// Mitsubishi GX Works2 project: EexcB-group13-1 (1) (1)   PLC: FX3G

// global labels: Global1
VAR_GLOBAL
  Switch7 AT X007 : BOOL;
  WorkLight AT Y007 : BOOL;
  Emergency_button AT X005 : BOOL;
  RaspberryStock AT D1100 : REAL;
  RaspberryInput AT D1110 : REAL;
  LemonStock AT D1102 : REAL;
  LemonInput AT D1112 : REAL;
  GummyBearStock AT D1104 : REAL;
  GummyBearInput AT D1114 : REAL;
  StablilizingMaterialStock AT D1106 : REAL;
  StablilizingMaterialInput AT D1116 : REAL;
  ANALOG_INPUT AT D8280 : INT;
  Intialize_produce AT X001 : BOOL;
  REGULAR_ICECREAM AT M0 : BOOL;
  ICE_CREAM_TYPE AT D1108 : REAL;
  UNDER_5 AT M2 : BOOL;
  UPPER_0 AT M3 : BOOL;
  UNDER_10 AT M4 : BOOL;
  UPPER_6 AT M6 : BOOL;
  PINUK_ICECREAM AT M1 : BOOL;
  LEMON_PINUK AT M11 : BOOL;
  RASPBERRY_PINUK AT M12 : BOOL;
  StABILIZE_PINUK AT M13 : BOOL;
  GUMMYBEAR_PINUK AT M14 : BOOL;
  RASPBERRY_REGUKAR AT M15 : BOOL;
  LEMON_REGULAR AT M16 : BOOL;
  StABILIZE_REGULAR AT M17 : BOOL;
  GUMMYBEAR_REGULAR AT M18 : BOOL;
  ICECREAM_APPROVE AT M19 : BOOL;
  TIMER_LIGHT_MIX AT TC0 : BOOL;
  LIGHT_TIMER_SWITCH AT TS0 : BOOL;
  LIGHT_TIMER_SWITCH_Y0 AT TS0 : BOOL;
  MAKING_LIGHT AT Y000 : BOOL;
  MAKING_TIMER_SWITCH_Y0 AT TS0 : BOOL;
  MAKING_TIMER AT TC0 : BOOL;
  MAKING_PROCESS AT M30 : BOOL;
  MOVE_TO_FREEZE_SWITCH AT X002 : BOOL;
  LEMON_MAKE_CONTAINER AT M21 : BOOL;
  RASPBERRY_MAKE_CONTAINER AT M22 : BOOL;
  FREEZE_LIGHT AT Y002 : BOOL;
  FREEZE_process AT M25 : BOOL;
  FREEZING_TIMER AT TC1 : BOOL;
  SENSOR_10 AT X003 : BOOL;
  FREEZING_TIMER_SWITCH AT TS1 : BOOL;
  FREEZE_DONE AT M26 : BOOL;
  MIX_PROCESS AT M26 : BOOL;
  MIX_CONTAINER AT M27 : BOOL;
  PINUK_MIX_TIMER AT TC2 : BOOL;
  REGULAR_MIX_TIMER AT TC3 : BOOL;
  PINUK_MIX_SWITCH AT TS2 : BOOL;
  REGULAR_MIX_SWITCH AT TS3 : BOOL;
  START_MIX AT M28 : BOOL;
  MIX_LIGHT_TIMER_1 AT TC4 : BOOL;
  MIX_LIGHT_SWITCH_1 AT TS4 : BOOL;
  BLINK_ENABLE AT M29 : BOOL;
  MIX_LIGHT_TIMER_2 AT TC5 : BOOL;
  MIX_LIGHT_SWITCH_2 AT TS5 : BOOL;
  TYPE_CHOSEN AT M10 : BOOL;
  ICECREAM_counter AT CC0 : BOOL;
  ICECREAM_READY AT M31 : BOOL;
  PROCESS_DONE AT M32 : BOOL;
  ANALOG_OUTPUT AT D8282 : INT;
  Sop AT M33 : BOOL;
  OUT_OF_STOCK AT M5 : BOOL;
  UNDER_6 AT M34 : BOOL;
  UPPER_5 AT M35 : BOOL;
  BLINK_LIGHT_1 AT Y005 : BOOL;
  BLINK_LIGHT_2 AT Y006 : BOOL;
  DELETE AT X030 : BOOL;
  InVENTORY_CHECK AT M36 : BOOL;
  OUT_OF_RAS AT M37 : BOOL;
  OUT_OF_LEMON AT M38 : BOOL;
  OUT_OF_STABILIZE AT M39 : BOOL;
  OUT_OF_GUMMY AT M40 : BOOL;
  InVENTORY_CHECK_DONE AT M41 : BOOL;
  ICE_CREAM_packs AT D1118 : REAL;
  RASPBERRY_ICECREAM_MAK_CONTAINER AT D1122 : REAL;
  LEMON_ICECREAM_MAK_CONTAINER AT D1120 : REAL;
  LEMON_FREEZE_CONTAINERR AT D1124 : REAL;
  RASPBERRY_FREEZE_CONTAINERR AT D1126 : REAL;
  MIXING_CONTAINER AT D1128 : REAL;
  MOVED_CONTAINER_2 AT M42 : BOOL;
  FINISHED_MOVE_2 AT M43 : BOOL;
  MOVE_CONTAINAER_2 AT TC6 : BOOL;
  FINISH_MOVING_2 AT TS6 : BOOL;
END_VAR

// task Task_01 (event TRUE, interval 0, priority 31): POU_01

PROGRAM POU_01
(* structured ladder/FBD written out as ST: instructions are called as NAME(EN, inputs, outputs); _pN, _eN, _tN stand for wires *)
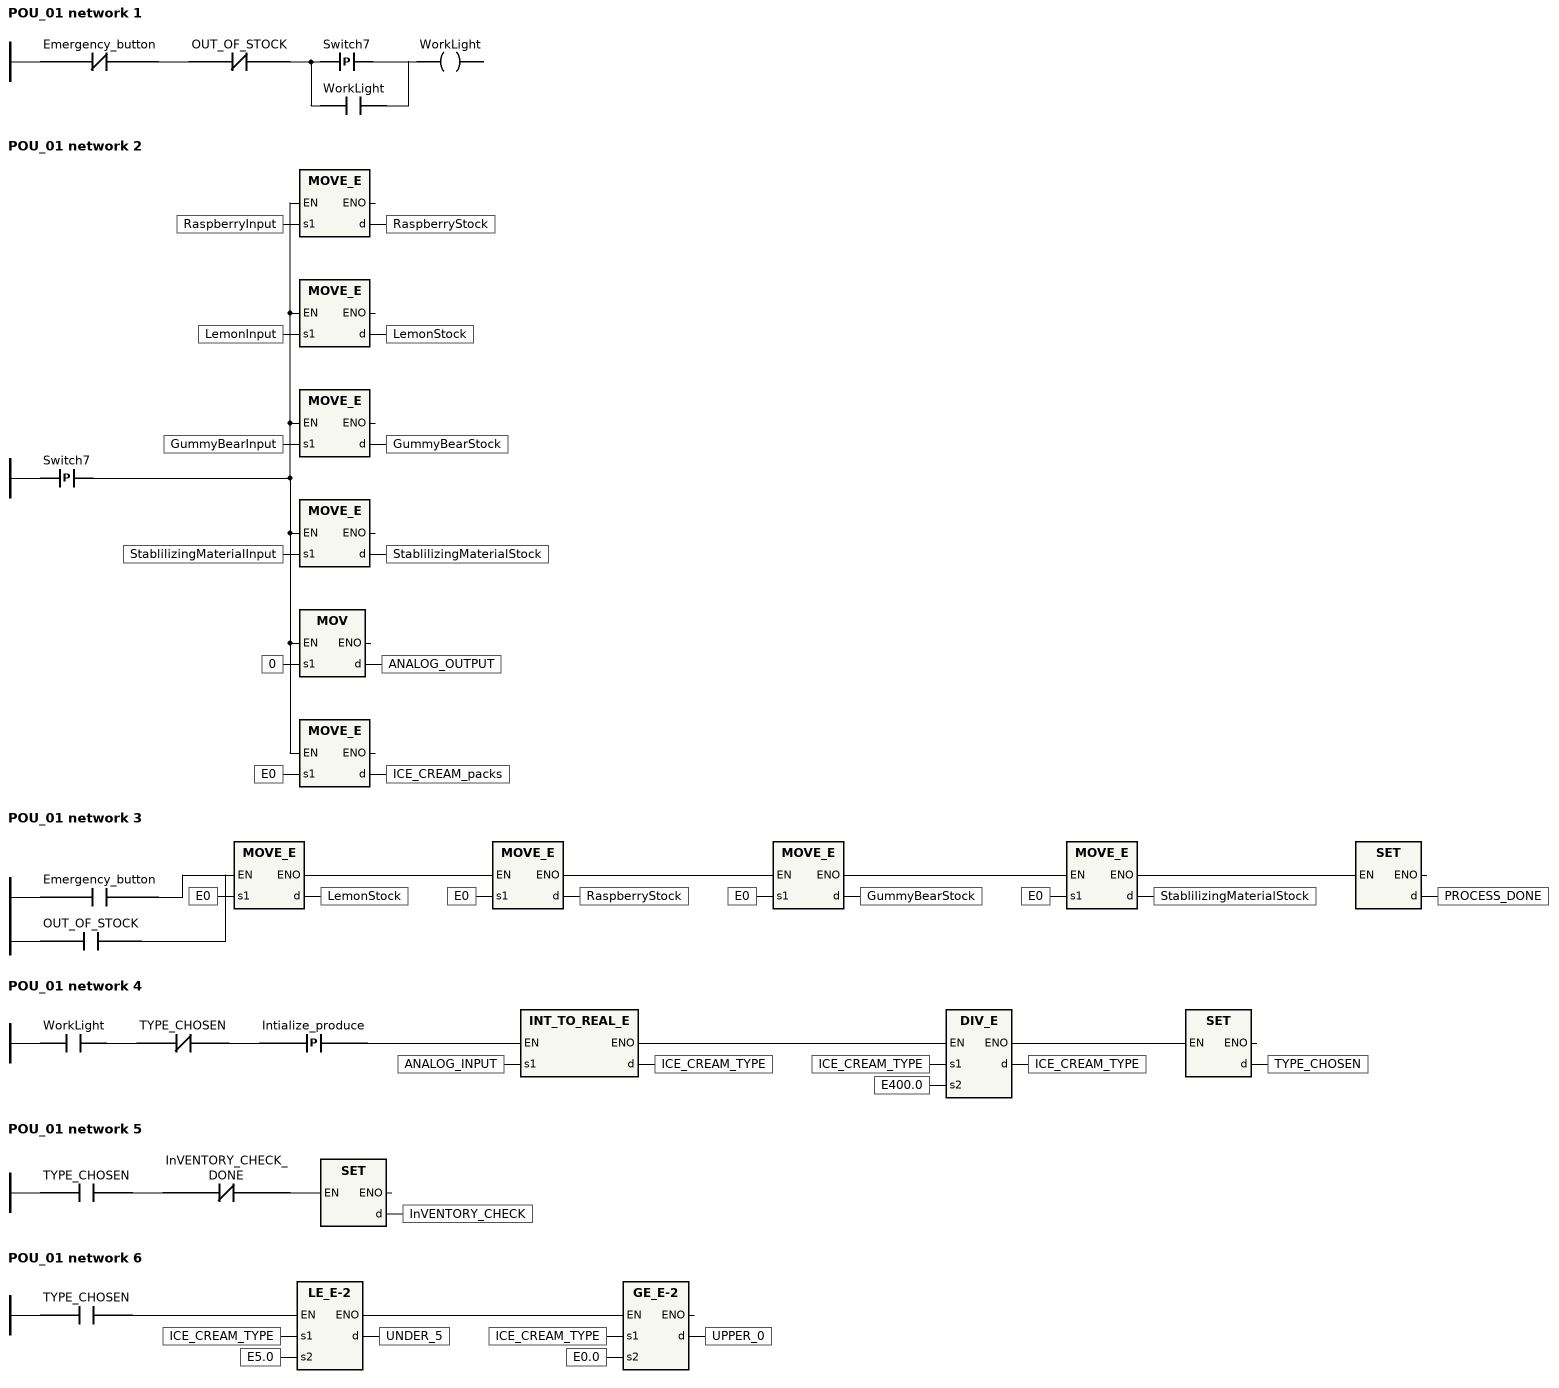
(* network 1 *)
_p1 := NOT Emergency_button AND NOT OUT_OF_STOCK;
WorkLight := (_p1 AND LDP(TRUE, Switch7)) OR (_p1 AND WorkLight);
(* network 2 *)
_p1 := LDP(TRUE, Switch7);
MOVE_E(_p1, RaspberryInput, RaspberryStock);
MOVE_E(_p1, LemonInput, LemonStock);
MOVE_E(_p1, GummyBearInput, GummyBearStock);
MOVE_E(_p1, StablilizingMaterialInput, StablilizingMaterialStock);
MOV(_p1, 0, ANALOG_OUTPUT);
MOVE_E(_p1, E0, ICE_CREAM_packs);
(* network 3 *)
_e1 := MOVE_E(Emergency_button OR OUT_OF_STOCK, E0, LemonStock);
_e2 := MOVE_E(_e1, E0, RaspberryStock);
_e3 := MOVE_E(_e2, E0, GummyBearStock);
_e4 := MOVE_E(_e3, E0, StablilizingMaterialStock);
SET(_e4, PROCESS_DONE);
(* network 4 *)
_e1 := INT_TO_REAL_E(WorkLight AND NOT TYPE_CHOSEN AND LDP(TRUE, Intialize_produce), ANALOG_INPUT, ICE_CREAM_TYPE);
_e2 := DIV_E(_e1, ICE_CREAM_TYPE, E400.0, ICE_CREAM_TYPE);
SET(_e2, TYPE_CHOSEN);
(* network 5 *)
SET(TYPE_CHOSEN AND NOT InVENTORY_CHECK_DONE, InVENTORY_CHECK);
(* network 6 *)
_e1 := LE_E(TYPE_CHOSEN, ICE_CREAM_TYPE, E5.0, UNDER_5);
GE_E(_e1, ICE_CREAM_TYPE, E0.0, UPPER_0);
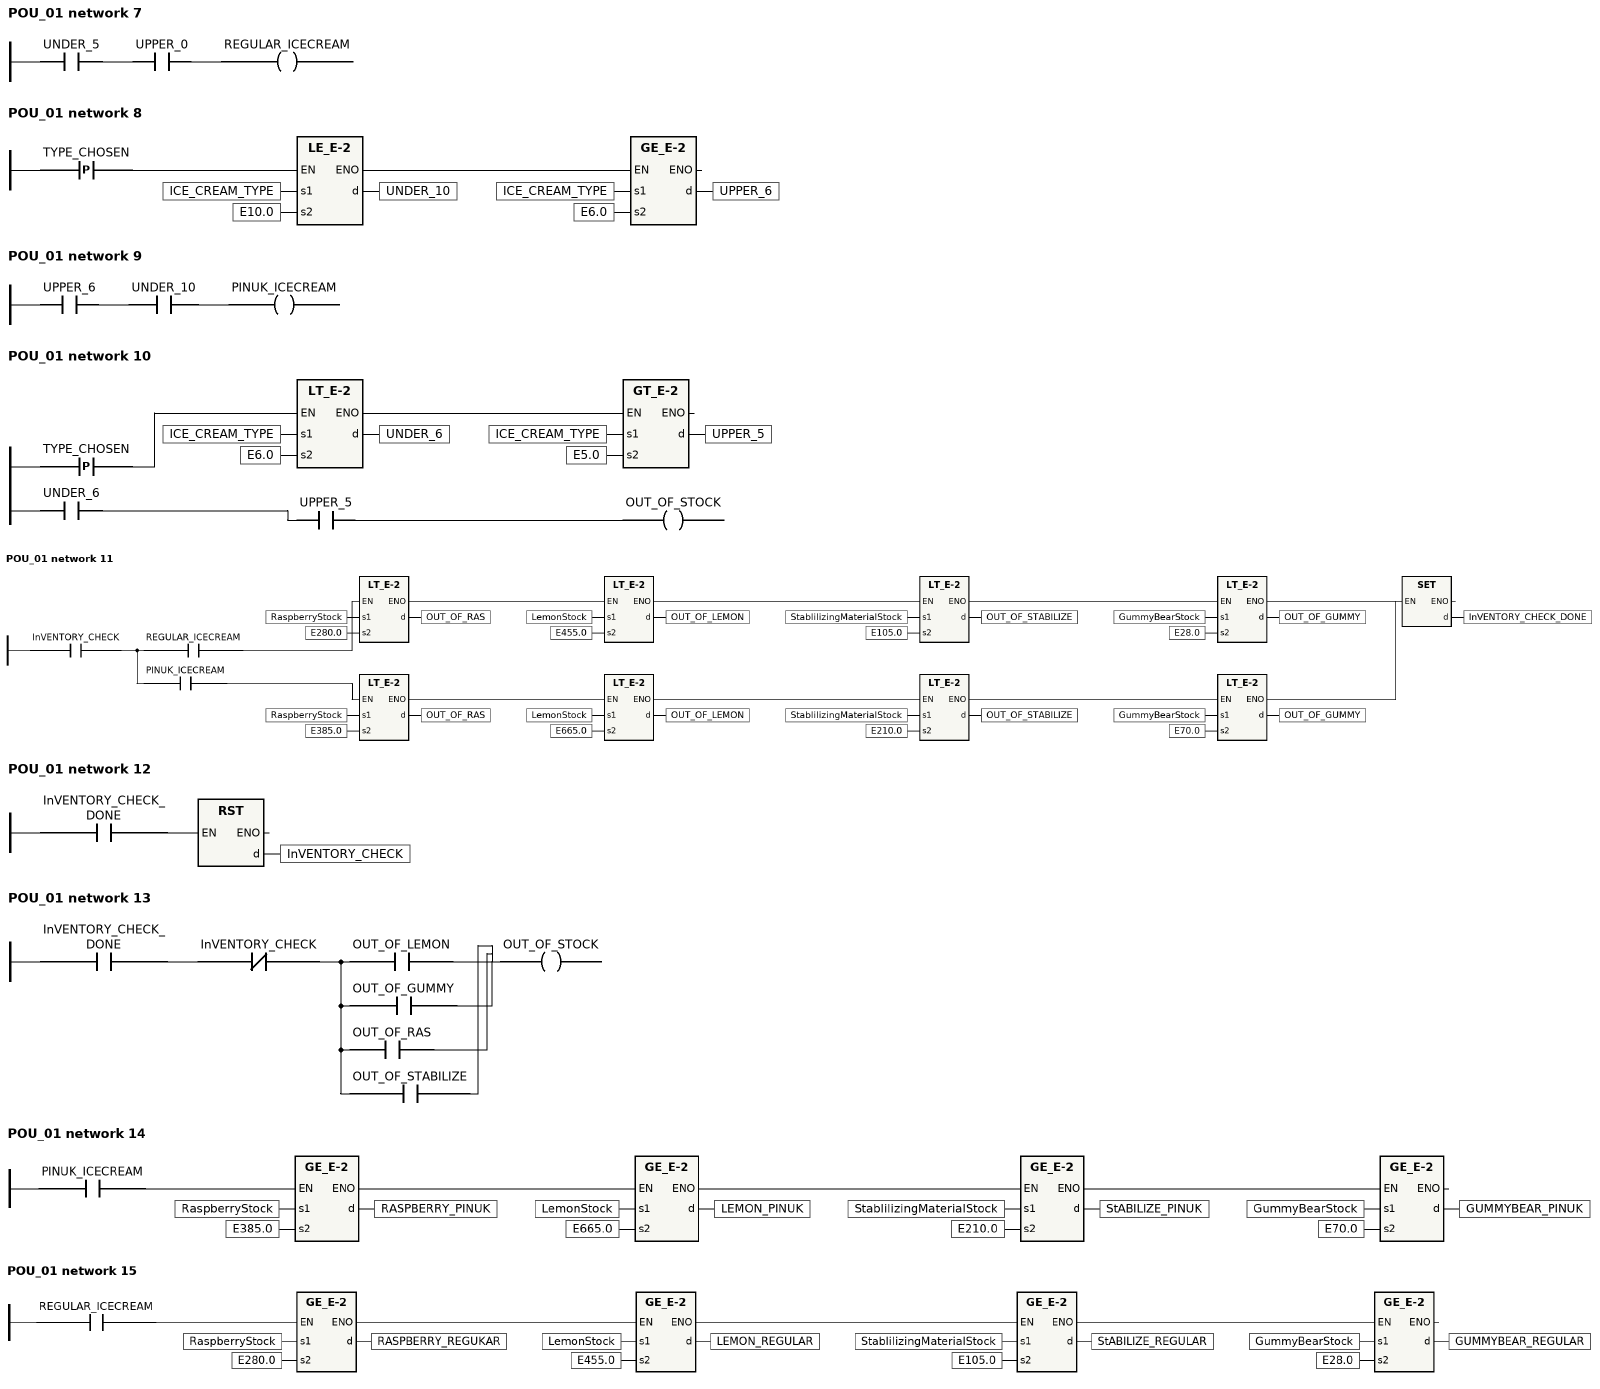
(* network 7 *)
REGULAR_ICECREAM := UNDER_5 AND UPPER_0;
(* network 8 *)
_e1 := LE_E(LDP(TRUE, TYPE_CHOSEN), ICE_CREAM_TYPE, E10.0, UNDER_10);
GE_E(_e1, ICE_CREAM_TYPE, E6.0, UPPER_6);
(* network 9 *)
PINUK_ICECREAM := UPPER_6 AND UNDER_10;
(* network 10 *)
_e1 := LT_E(LDP(TRUE, TYPE_CHOSEN), ICE_CREAM_TYPE, E6.0, UNDER_6);
GT_E(_e1, ICE_CREAM_TYPE, E5.0, UPPER_5);
OUT_OF_STOCK := UNDER_6 AND UPPER_5;
(* network 11 *)
_e1 := LT_E(InVENTORY_CHECK AND REGULAR_ICECREAM, RaspberryStock, E280.0, OUT_OF_RAS);
_e2 := LT_E(_e1, LemonStock, E455.0, OUT_OF_LEMON);
_e3 := LT_E(_e2, StablilizingMaterialStock, E105.0, OUT_OF_STABILIZE);
_e4 := LT_E(_e3, GummyBearStock, E28.0, OUT_OF_GUMMY);
_e5 := LT_E(InVENTORY_CHECK AND PINUK_ICECREAM, RaspberryStock, E385.0, OUT_OF_RAS);
_e6 := LT_E(_e5, LemonStock, E665.0, OUT_OF_LEMON);
_e7 := LT_E(_e6, StablilizingMaterialStock, E210.0, OUT_OF_STABILIZE);
_e8 := LT_E(_e7, GummyBearStock, E70.0, OUT_OF_GUMMY);
SET(_e4 OR _e8, InVENTORY_CHECK_DONE);
(* network 12 *)
RST(InVENTORY_CHECK_DONE, InVENTORY_CHECK);
(* network 13 *)
_p1 := InVENTORY_CHECK_DONE AND NOT InVENTORY_CHECK;
OUT_OF_STOCK := (_p1 AND OUT_OF_LEMON) OR (_p1 AND OUT_OF_GUMMY) OR (_p1 AND OUT_OF_RAS) OR (_p1 AND OUT_OF_STABILIZE);
(* network 14 *)
_e1 := GE_E(PINUK_ICECREAM, RaspberryStock, E385.0, RASPBERRY_PINUK);
_e2 := GE_E(_e1, LemonStock, E665.0, LEMON_PINUK);
_e3 := GE_E(_e2, StablilizingMaterialStock, E210.0, StABILIZE_PINUK);
GE_E(_e3, GummyBearStock, E70.0, GUMMYBEAR_PINUK);
(* network 15 *)
_e1 := GE_E(REGULAR_ICECREAM, RaspberryStock, E280.0, RASPBERRY_REGUKAR);
_e2 := GE_E(_e1, LemonStock, E455.0, LEMON_REGULAR);
_e3 := GE_E(_e2, StablilizingMaterialStock, E105.0, StABILIZE_REGULAR);
GE_E(_e3, GummyBearStock, E28.0, GUMMYBEAR_REGULAR);
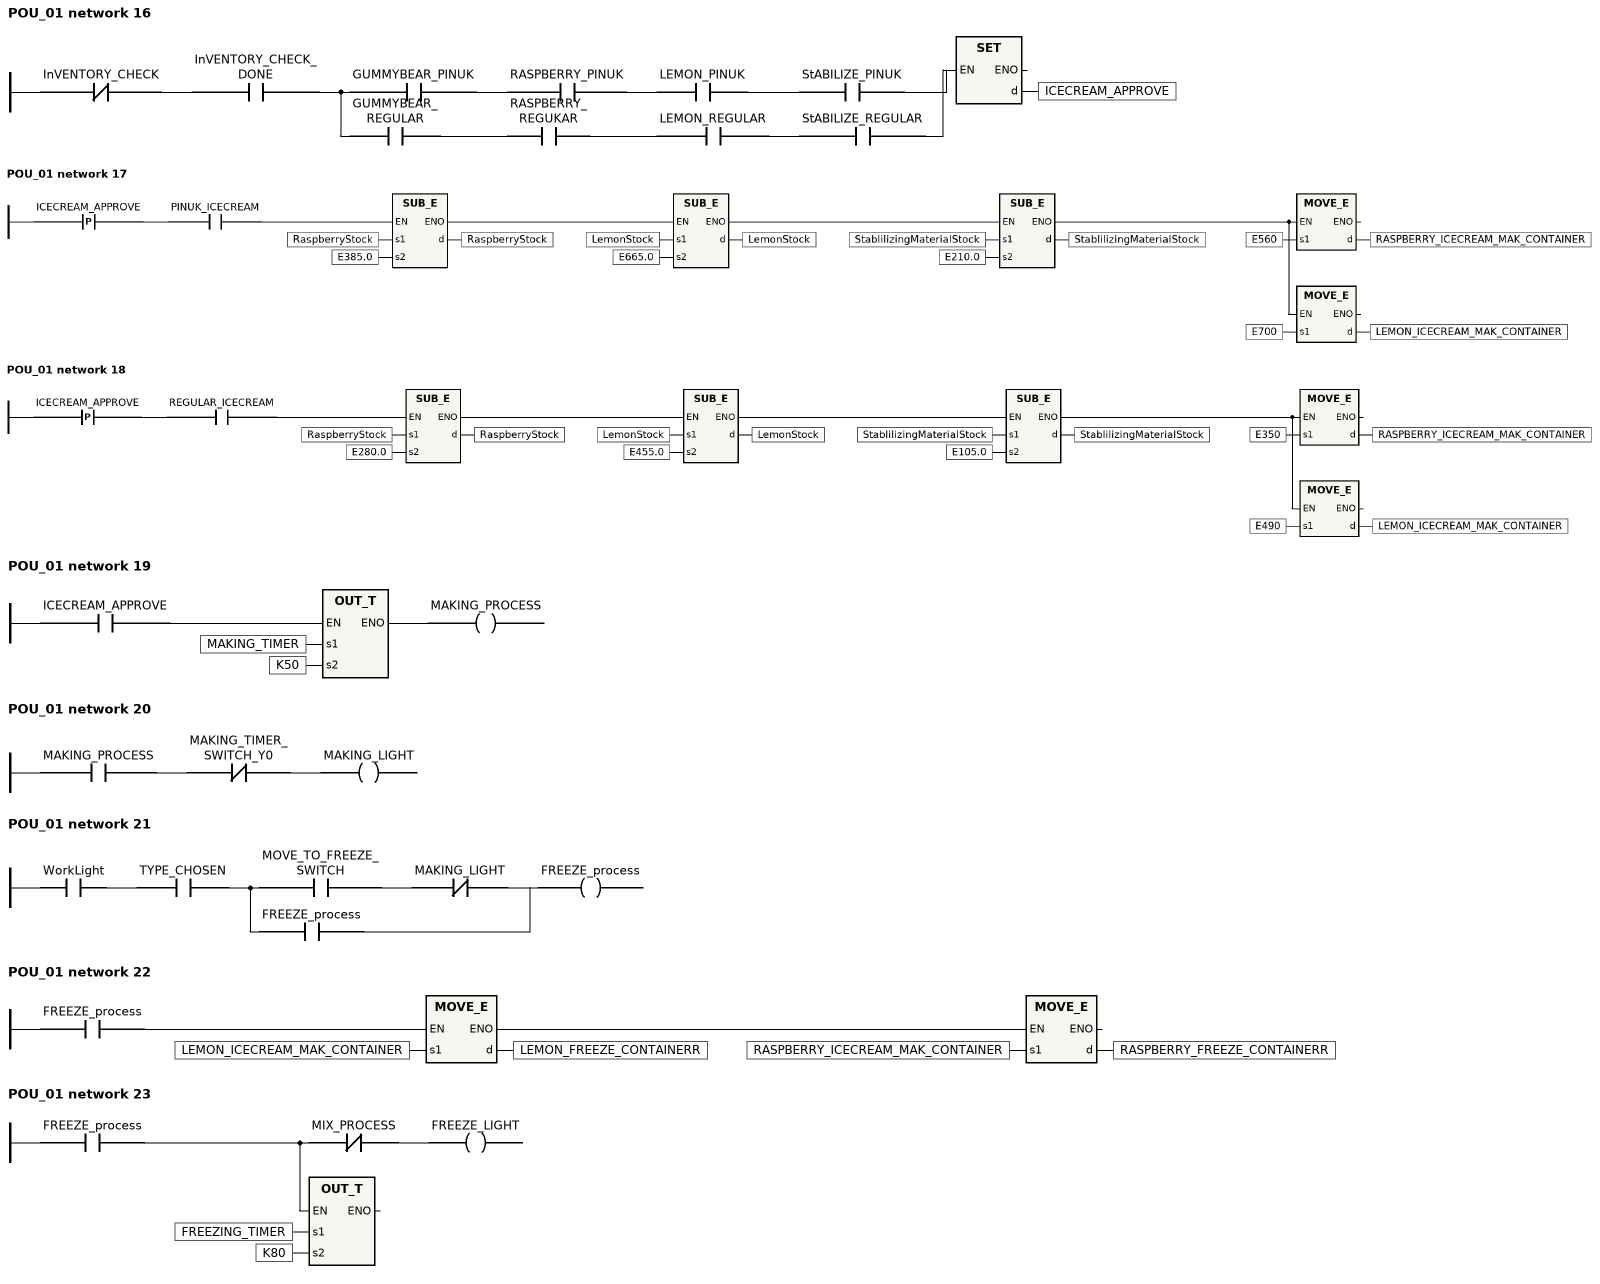
(* network 16 *)
_p1 := NOT InVENTORY_CHECK AND InVENTORY_CHECK_DONE;
SET((_p1 AND GUMMYBEAR_PINUK AND RASPBERRY_PINUK AND LEMON_PINUK AND StABILIZE_PINUK) OR (_p1 AND GUMMYBEAR_REGULAR AND RASPBERRY_REGUKAR AND LEMON_REGULAR AND StABILIZE_REGULAR), ICECREAM_APPROVE);
(* network 17 *)
_e1 := SUB_E(LDP(TRUE, ICECREAM_APPROVE) AND PINUK_ICECREAM, RaspberryStock, E385.0, RaspberryStock);
_e2 := SUB_E(_e1, LemonStock, E665.0, LemonStock);
_e3 := SUB_E(_e2, StablilizingMaterialStock, E210.0, StablilizingMaterialStock);
MOVE_E(_e3, E560, RASPBERRY_ICECREAM_MAK_CONTAINER);
MOVE_E(_e3, E700, LEMON_ICECREAM_MAK_CONTAINER);
(* network 18 *)
_e1 := SUB_E(LDP(TRUE, ICECREAM_APPROVE) AND REGULAR_ICECREAM, RaspberryStock, E280.0, RaspberryStock);
_e2 := SUB_E(_e1, LemonStock, E455.0, LemonStock);
_e3 := SUB_E(_e2, StablilizingMaterialStock, E105.0, StablilizingMaterialStock);
MOVE_E(_e3, E350, RASPBERRY_ICECREAM_MAK_CONTAINER);
MOVE_E(_e3, E490, LEMON_ICECREAM_MAK_CONTAINER);
(* network 19 *)
_e1 := OUT_T(ICECREAM_APPROVE, MAKING_TIMER, K50);
MAKING_PROCESS := _e1;
(* network 20 *)
MAKING_LIGHT := MAKING_PROCESS AND NOT MAKING_TIMER_SWITCH_Y0;
(* network 21 ICECREAM_FREEZE *)
_p1 := WorkLight AND TYPE_CHOSEN;
FREEZE_process := (_p1 AND MOVE_TO_FREEZE_SWITCH AND NOT MAKING_LIGHT) OR (_p1 AND FREEZE_process);
(* network 22 *)
_e1 := MOVE_E(FREEZE_process, LEMON_ICECREAM_MAK_CONTAINER, LEMON_FREEZE_CONTAINERR);
MOVE_E(_e1, RASPBERRY_ICECREAM_MAK_CONTAINER, RASPBERRY_FREEZE_CONTAINERR);
(* network 23 *)
FREEZE_LIGHT := FREEZE_process AND NOT MIX_PROCESS;
OUT_T(FREEZE_process, FREEZING_TIMER, K80);
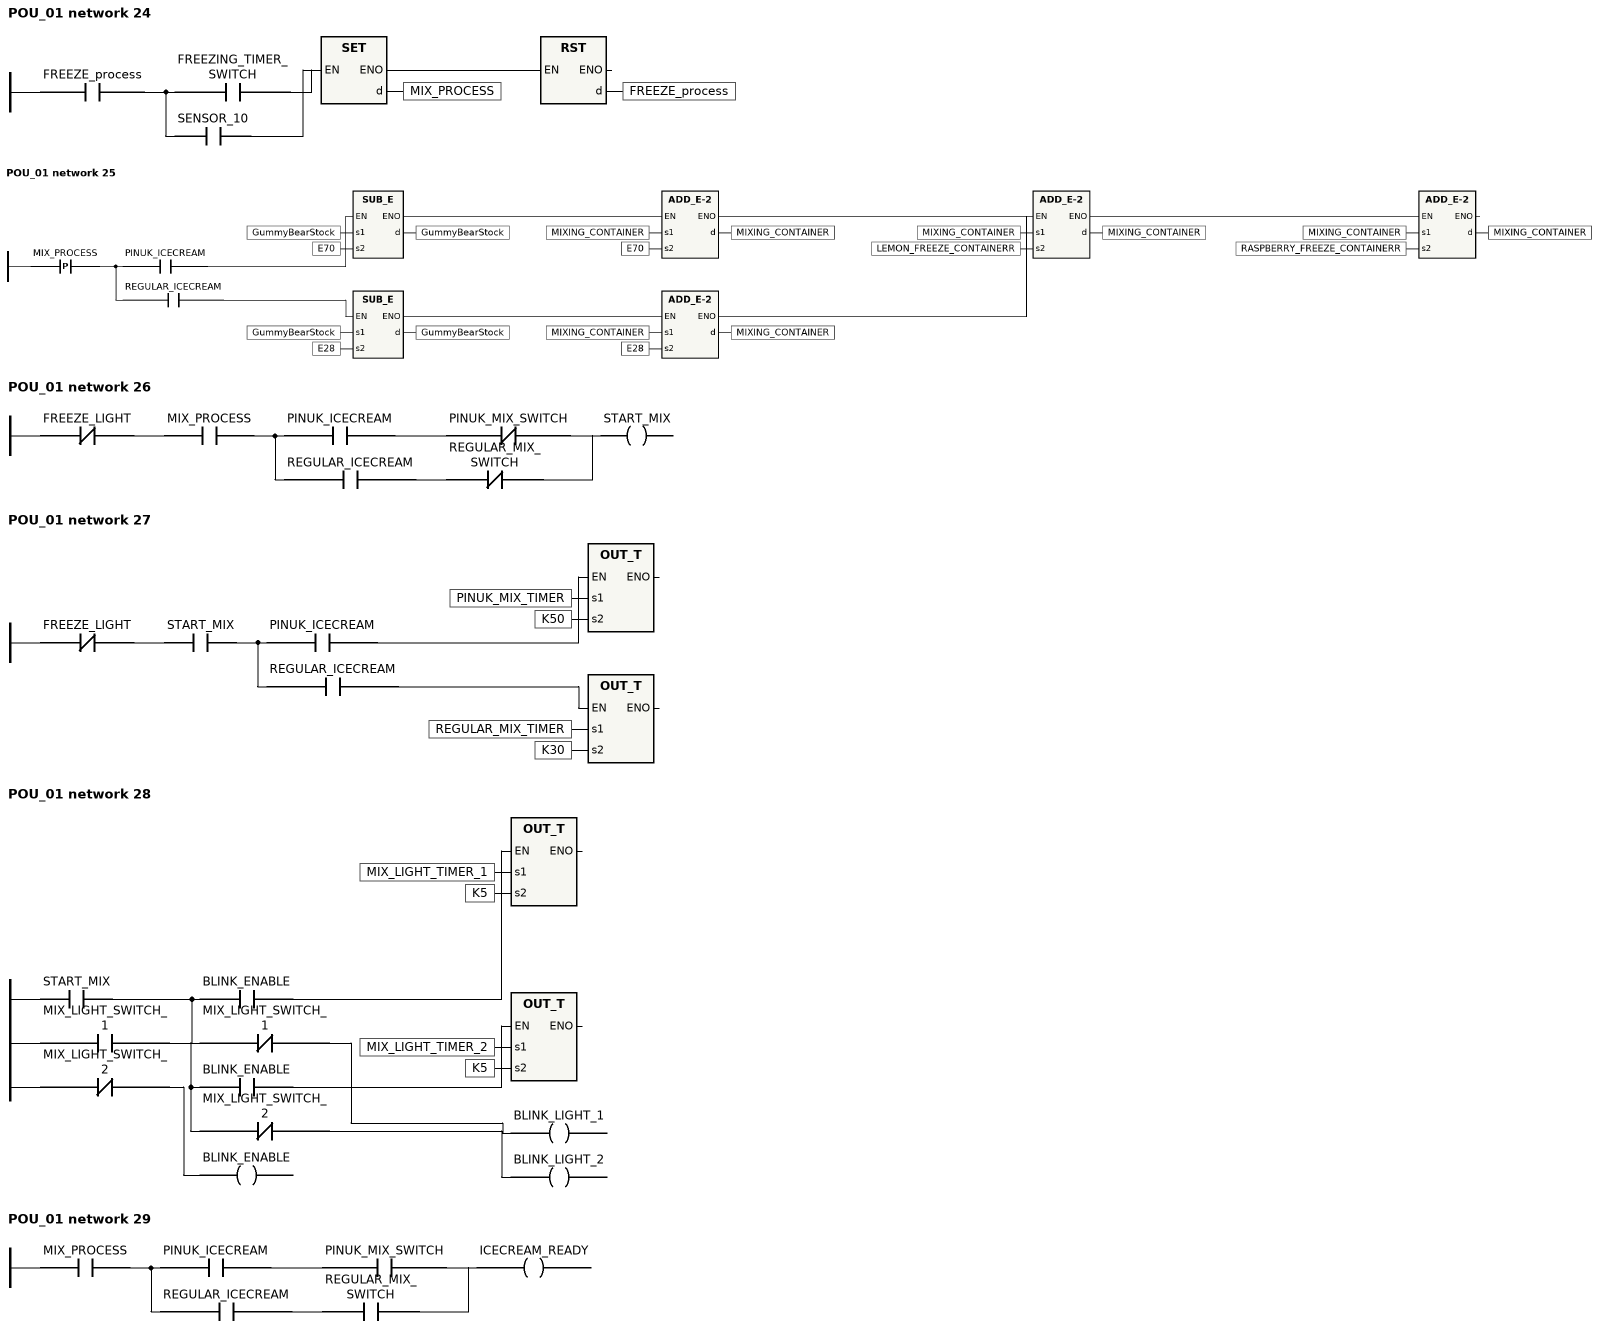
(* network 24 *)
_e1 := SET((FREEZE_process AND FREEZING_TIMER_SWITCH) OR (FREEZE_process AND SENSOR_10), MIX_PROCESS);
RST(_e1, FREEZE_process);
(* network 25 *)
_p1 := LDP(TRUE, MIX_PROCESS);
_e2 := SUB_E(_p1 AND PINUK_ICECREAM, GummyBearStock, E70, GummyBearStock);
_e3 := ADD_E(_e2, MIXING_CONTAINER, E70, MIXING_CONTAINER);
_e4 := SUB_E(_p1 AND REGULAR_ICECREAM, GummyBearStock, E28, GummyBearStock);
_e5 := ADD_E(_e4, MIXING_CONTAINER, E28, MIXING_CONTAINER);
_e6 := ADD_E(_e3 OR _e5, MIXING_CONTAINER, LEMON_FREEZE_CONTAINERR, MIXING_CONTAINER);
ADD_E(_e6, MIXING_CONTAINER, RASPBERRY_FREEZE_CONTAINERR, MIXING_CONTAINER);
(* network 26 *)
_p1 := NOT FREEZE_LIGHT AND MIX_PROCESS;
START_MIX := (_p1 AND PINUK_ICECREAM AND NOT PINUK_MIX_SWITCH) OR (_p1 AND REGULAR_ICECREAM AND NOT REGULAR_MIX_SWITCH);
(* network 27 *)
_p1 := NOT FREEZE_LIGHT AND START_MIX;
OUT_T(_p1 AND PINUK_ICECREAM, PINUK_MIX_TIMER, K50);
OUT_T(_p1 AND REGULAR_ICECREAM, REGULAR_MIX_TIMER, K30);
(* network 28 *)
OUT_T(START_MIX AND BLINK_ENABLE, MIX_LIGHT_TIMER_1, K5);
BLINK_LIGHT_1 := START_MIX AND NOT MIX_LIGHT_SWITCH_1;
OUT_T(MIX_LIGHT_SWITCH_1 AND BLINK_ENABLE, MIX_LIGHT_TIMER_2, K5);
BLINK_LIGHT_2 := MIX_LIGHT_SWITCH_1 AND NOT MIX_LIGHT_SWITCH_2;
BLINK_ENABLE := NOT MIX_LIGHT_SWITCH_2;
(* network 29 *)
ICECREAM_READY := (MIX_PROCESS AND PINUK_ICECREAM AND PINUK_MIX_SWITCH) OR (MIX_PROCESS AND REGULAR_ICECREAM AND REGULAR_MIX_SWITCH);
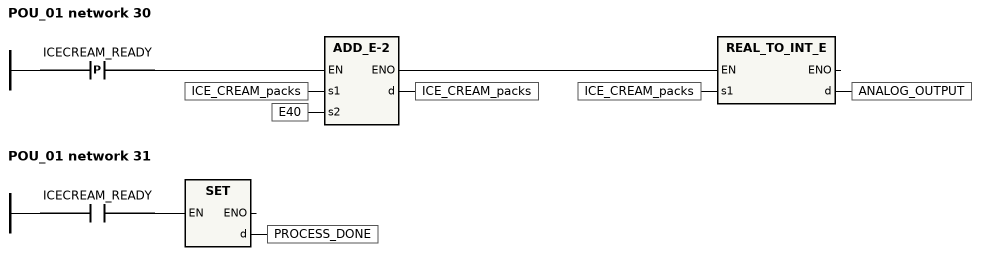
(* network 30 *)
_e1 := ADD_E(LDP(TRUE, ICECREAM_READY), ICE_CREAM_packs, E40, ICE_CREAM_packs);
REAL_TO_INT_E(_e1, ICE_CREAM_packs, ANALOG_OUTPUT);
(* network 31 *)
SET(ICECREAM_READY, PROCESS_DONE);
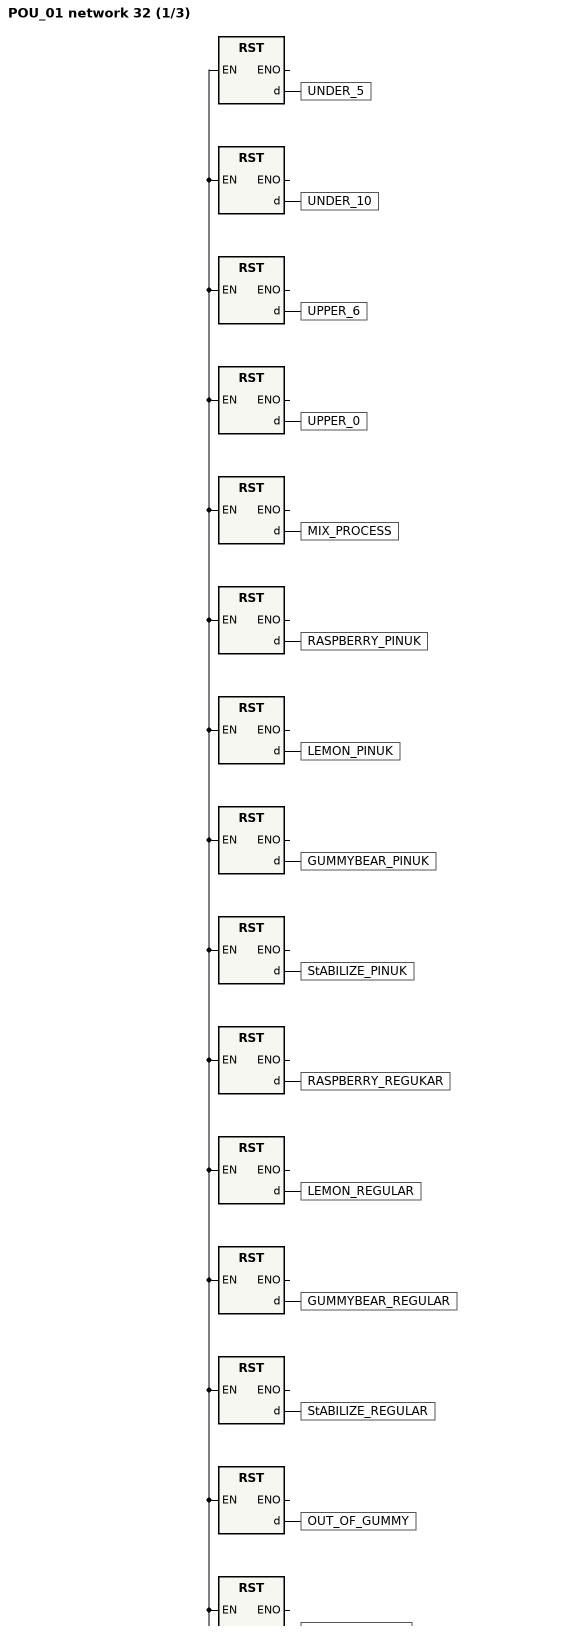
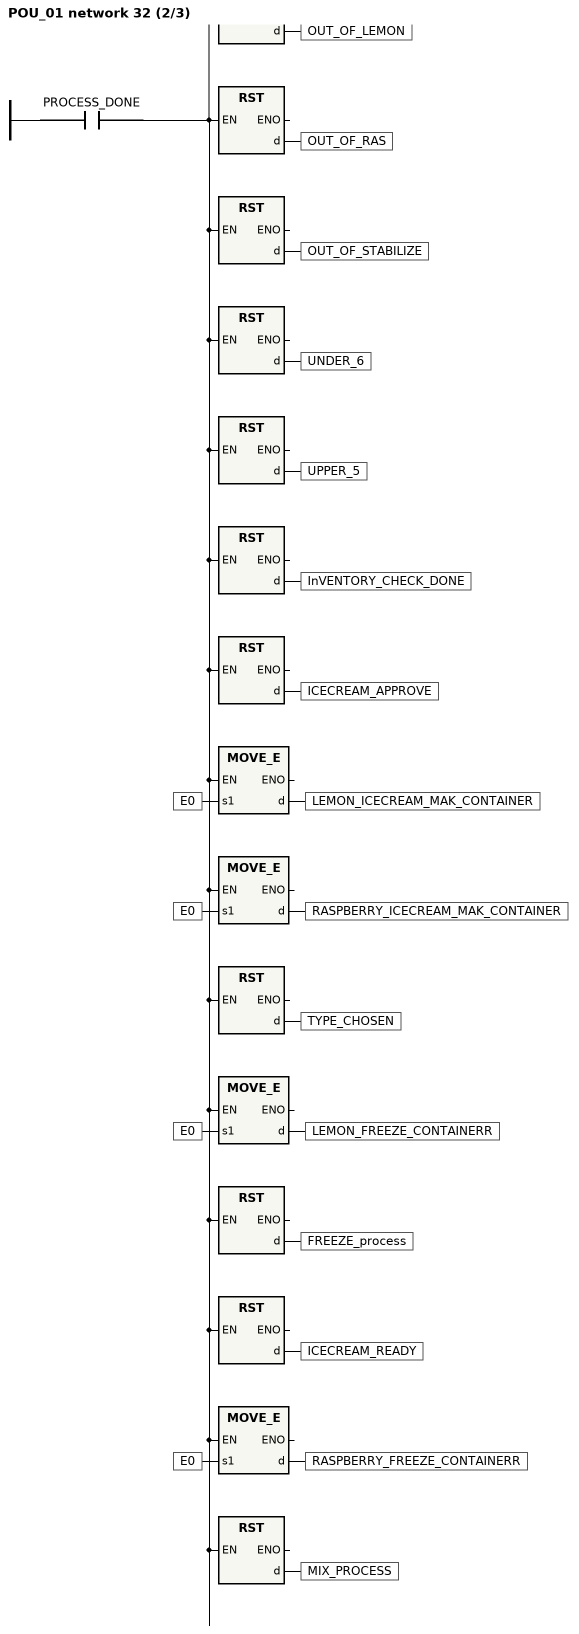
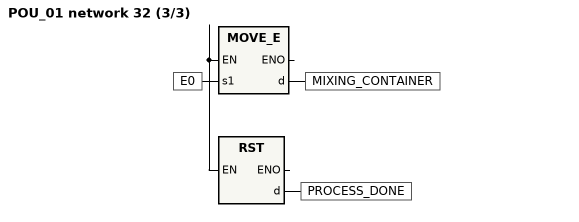
(* network 32 *)
RST(PROCESS_DONE, UNDER_5);
RST(PROCESS_DONE, UNDER_10);
RST(PROCESS_DONE, UPPER_6);
RST(PROCESS_DONE, UPPER_0);
RST(PROCESS_DONE, MIX_PROCESS);
RST(PROCESS_DONE, RASPBERRY_PINUK);
RST(PROCESS_DONE, LEMON_PINUK);
RST(PROCESS_DONE, GUMMYBEAR_PINUK);
RST(PROCESS_DONE, StABILIZE_PINUK);
RST(PROCESS_DONE, RASPBERRY_REGUKAR);
RST(PROCESS_DONE, LEMON_REGULAR);
RST(PROCESS_DONE, GUMMYBEAR_REGULAR);
RST(PROCESS_DONE, StABILIZE_REGULAR);
RST(PROCESS_DONE, OUT_OF_GUMMY);
RST(PROCESS_DONE, OUT_OF_LEMON);
RST(PROCESS_DONE, OUT_OF_RAS);
RST(PROCESS_DONE, OUT_OF_STABILIZE);
RST(PROCESS_DONE, UNDER_6);
RST(PROCESS_DONE, UPPER_5);
RST(PROCESS_DONE, InVENTORY_CHECK_DONE);
RST(PROCESS_DONE, ICECREAM_APPROVE);
MOVE_E(PROCESS_DONE, E0, LEMON_ICECREAM_MAK_CONTAINER);
MOVE_E(PROCESS_DONE, E0, RASPBERRY_ICECREAM_MAK_CONTAINER);
RST(PROCESS_DONE, TYPE_CHOSEN);
MOVE_E(PROCESS_DONE, E0, LEMON_FREEZE_CONTAINERR);
RST(PROCESS_DONE, FREEZE_process);
RST(PROCESS_DONE, ICECREAM_READY);
MOVE_E(PROCESS_DONE, E0, RASPBERRY_FREEZE_CONTAINERR);
RST(PROCESS_DONE, MIX_PROCESS);
MOVE_E(PROCESS_DONE, E0, MIXING_CONTAINER);
RST(PROCESS_DONE, PROCESS_DONE);
END_PROGRAM
